{attribute 'linkalways'} 
{attribute 'no_explicit_call' := 'This FB is a CLASS and must be accessed using methods or properties'}
{attribute 'enable_dynamic_creation'}
FUNCTION_BLOCK Node_F_VN_InsertIntoContainer_TcVnPoint2_REAL EXTENDS VisionNode
VAR
    aElement : _TcVnPoint2_REAL;
    ipContainer : _ITcVnContainer;
    nIndex : _ULINT(0);
    hrPrev : _HRESULT(S_OK);
    hresult : _HRESULT(S_OK);
END_VAR

METHOD PUBLIC  Clone : I_Node
VAR
	pNode : POINTER TO Node_F_VN_InsertIntoContainer_TcVnPoint2_REAL;
END_VAR
pNode := __NEW(Node_F_VN_InsertIntoContainer_TcVnPoint2_REAL);
Clone := pNode^;
END_METHOD

METHOD FB_init : BOOL
VAR_INPUT
	bInitRetains : BOOL; // if TRUE, the retain variables are initialized (warm start / cold start)
	bInCopyCode : BOOL;  // if TRUE, the instance afterwards gets moved into the copy code (online change)
END_VAR
AddInput('aElement', aElement);
AddInput('ipContainer', ipContainer);
AddInput('nIndex', nIndex);
AddInput('hrPrev', hrPrev);
AddOutput('ipContainer', ipContainer);
AddOutput('hresult',hresult);
END_METHOD

METHOD PROTECTED OnExecute : HRESULT
hresult.Value := F_VN_InsertIntoContainer_TcVnPoint2_REAL(
    aElement := aElement.Value,
    ipContainer := ipContainer.Value,
    nIndex := nIndex.Value,
    hrPrev:= hrPrev.Value);
END_METHOD

METHOD PUBLIC PreExecutionCheck
VAR_INPUT
	Check : I_PreExecutionChecks;
END_VAR
Check.IsTrue(ipContainer.IsValid, 'ipContainer must be a valid container');
END_METHOD

END_FUNCTION_BLOCK

(* stored: Version 1.1.0.1, ProductVersion 3.1.4024.13
   POU Node_F_VN_InsertIntoContainer_TcVnPoint2_REAL: Id {03e00115-da9c-4c9b-a4a0-2995bc9e7158}, SpecialFunc None
   Folder Constructor: Id {f4067b4a-262e-49af-bba1-4d89855ae540}
   Method Clone: Id {b19cb71b-0fa5-4a19-8bec-f00a36044882}
   Method FB_init: Id {9c24bc75-9a8c-4371-964f-282fbdeeb3a2}
   Method OnExecute: Id {1e2709c2-0d30-4c10-973e-57ec54152af1}
   Method PreExecutionCheck: Id {7bbebe7a-f537-4f16-8f33-d8e39c335c2f} *)
